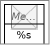
VISUALIZATION VISU_VANNE_2P_H  // 50x45
VAR_IN_OUT
	m_Input_VANNE : BLOCK_ACTUATOR;
END_VAR
    Rectangle (4,4 40x40), invisible if: TRUE
    Polygon (0,0)
    Rectangle (-1,25 50x20), "%s", text variable: m_Input_VANNE.MNEMO
    Polygon (0,0), colour toggle: (m_Input_VANNE.STATE_ON) <> 0, invisible if: NOT (m_Input_VANNE.STATE_OFF OR m_Input_VANNE.STATE_ON)
    Image (11,4 26x25), invisible if: NOT m_Input_VANNE.STATE_Nok, image: MesImages.warning
    Rectangle (4,4 40x20), invisible if: NOT (m_Input_VANNE.Autor_ON_IHM OR m_Input_VANNE.Autor_OFF_IHM) OR NOT PRG_User.ACTU_USER.MAINTENANCE
        tap m_Input_VANNE.M_ON
END_VISUALIZATION

(* stored: Version 1.1.0.1, ProductVersion 3.1.4024.12
   Visu VISU_VANNE_2P_H: Id {7bc2d8a3-3a3f-4aff-80be-55ffc45306f7} *)
